// Mitsubishi GX Works2 project: servo_extend_2   PLC: Q02/Q02H

PROGRAM MAIN
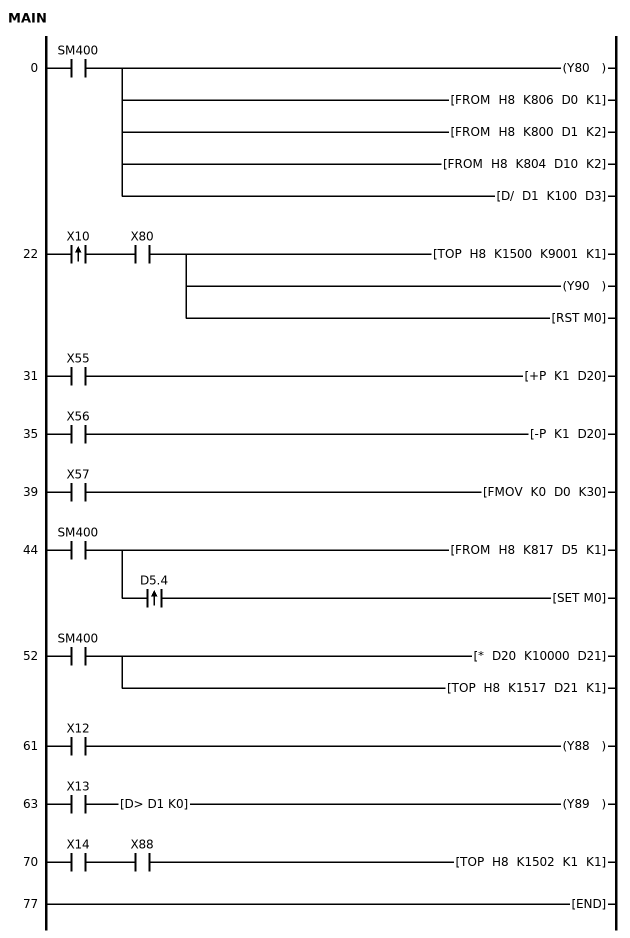
0     LD      SM400
      OUT     Y80
      FROM    H8 K806 D0 K1
      FROM    H8 K800 D1 K2
      FROM    H8 K804 D10 K2
      D/      D1 K100 D3
22    LDP     X10
      AND     X80
      TOP     H8 K1500 K9001 K1
      OUT     Y90
      RST     M0
31    LD      X55
      +P      K1 D20
35    LD      X56
      -P      K1 D20
39    LD      X57
      FMOV    K0 D0 K30
44    LD      SM400
      FROM    H8 K817 D5 K1
      ANDP    D5.4
      SET     M0
52    LD      SM400
      *       D20 K10000 D21
      TOP     H8 K1517 D21 K1
61    LD      X12
      OUT     Y88
63    LD      X13
      ANDD>   D1 K0
      OUT     Y89
70    LD      X14
      AND     X88
      TOP     H8 K1502 K1 K1
77    END
END_PROGRAM
